// TwinCAT 3 PLC project SquareWaveGenerator
// ProgramVersion: 3.1.4024.0
// libraries:
//   Tc2_Standard, * (Beckhoff Automation GmbH)
//   Tc2_System, * (Beckhoff Automation GmbH)
//   Tc3_Module, * (Beckhoff Automation GmbH)
//   VisuSymbols,3.5.10.0,System
// project tree:
//   / GlobalTextList.TcGTLO, PlcTask.TcTTO, Visualization Manager.TcVMO (not stored)
//   POUs/ FB_SquareWaveGenerator.TcPOU, MAIN.TcPOU
//   VISUs/ VisualizationSquareWaveGenerator.TcVIS
// real-time tasks:
//   TASK PlcTask: cycle T#10ms, priority 20, ADS port 350

CONFIGURATION SquareWaveGenerator
    RESOURCE PLC ON TwinCAT3
        TASK PlcTask(INTERVAL := T#10ms, PRIORITY := 20);
        PROGRAM MAIN WITH PlcTask : MAIN;
    END_RESOURCE
END_CONFIGURATION

// ---- POUs/MAIN.TcPOU
PROGRAM MAIN
VAR
	bStartStop: BOOL := FALSE;
	bPulse: BOOL := FALSE;
	
	fbSWG : FB_SquareWaveGenerator;
END_VAR
VAR CONSTANT
	HIGHTIME : TIME := T#2S;
	LOWTIME : TIME := T#3S;
END_VAR

fbSWG(
	bStartStop := bStartStop, 
	tHighTime := HIGHTIME,
	tLowTime := LOWTIME,
	bOutPulse => bPulse);

END_PROGRAM

// ---- POUs/FB_SquareWaveGenerator.TcPOU
FUNCTION_BLOCK PUBLIC FB_SquareWaveGenerator
VAR_INPUT
	bStartStop : BOOL;
	tHighTime : TIME := T#1S;
	tLowTime : TIME := T#1S;
END_VAR
VAR_OUTPUT
	bOutPulse: BOOL;
END_VAR
VAR
	fbTON : TON;
	eState: (NotStarted, Started);
	bTimerState: BOOL := FALSE;
	tDuration: TIME := tHighTime;
END_VAR

fbTON (IN:= bTimerState, PT:= tDuration);

CASE eState OF
	NotStarted:
		IF bStartStop THEN
			Start();
		END_IF
		
	Started:
		IF fbTON.Q THEN
			Toggle();
		END_IF
		
		IF NOT bStartStop THEN
			Stop();
		END_IF
END_CASE

METHOD PRIVATE Start : BOOL
eState := Started;
bOutPulse := TRUE;

tDuration := tHighTime;
bTimerState := TRUE;

Start := TRUE;
END_METHOD

METHOD PRIVATE Stop : BOOL
fbTON (IN := FALSE);

bTimerState := FALSE;
eState := NotStarted;
bOutPulse := FALSE;

Stop := TRUE;
END_METHOD

METHOD PRIVATE Toggle : BOOL
fbTON (IN := FALSE);

bOutPulse := NOT bOutPulse;
IF bOutPulse THEN
	tDuration := tHighTime;
ELSE
	tDuration := tLowTime;
END_IF
bTimerState := TRUE;

Toggle := TRUE;
END_METHOD

END_FUNCTION_BLOCK

// ---- VISUs/VisualizationSquareWaveGenerator.TcVIS
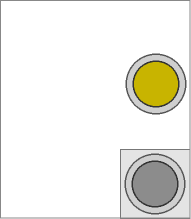
VISUALIZATION VisualizationSquareWaveGenerator  // 191x219
    PushSwitch (120,149 70x70), behaviour: TOGGLE, style: Switch-PushSwitch-Gray
    Lamp1 (121,49 70x70), variable: MAIN.bPulse, style: Lamp-Lamp1-Yellow
END_VISUALIZATION
